(* IEC 61131-3 sources: repolevel_ST_code_completion/dataset/project_code/ProductionLine/FUN, 6 files *)

(* ---- Motor.st ---- *)
FUNCTION_BLOCK Motor
VAR_INPUT
	MotorI:MotorI;
END_VAR
VAR_OUTPUT
	MotorO:MotorO;
END_VAR
VAR
	WaitTimer:TON;
	InternalSequenceDelay:time;
END_VAR

SetFault();
ResetFault();

(* ---- Motor_ResetFault.st ---- *)
METHOD ResetFault : BOOL
VAR_INPUT
	MotorI:MotorI;
END_VAR
VAR_OUTPUT
	MotorO:MotorO;
END_VAR
VAR
	WaitTimer:TON;
	InternalSequenceDelay:time;
	ResetDetect:r_trig;
END_VAR

ResetDetect(CLK:=MotorI.FaultReset);

IF ResetDetect.Q THEN
	MotorO.FaultStatus:=FALSE;
END_IF

(* ---- Motor_SetFault.st ---- *)
METHOD SetFault : BOOL
VAR_INPUT
	MotorI:MotorI;
END_VAR
VAR_OUTPUT
	MotorO:MotorO;
END_VAR
VAR
	WaitTimer:TON;
	InternalSequenceDelay:time;
END_VAR

IF MotorI.Overload THEN
	MotorO.FaultStatus:=TRUE;
	TurnOff();
END_IF

(* ---- Motor_SetWaitTime.st ---- *)
METHOD SetWaitTime : BOOL
VAR_INPUT
	MotorI:MotorI;
	SequenceDelay:TIME;
END_VAR
VAR_OUTPUT
	MotorO:MotorO;
END_VAR
VAR
	WaitTimer:TON;
	InternalSequenceDelay:time;
END_VAR

InternalSequenceDelay:=SequenceDelay;

(* ---- Motor_TurnOff.st ---- *)
METHOD TurnOff : BOOL
VAR_INPUT
	MotorI:MotorI;
END_VAR
VAR_OUTPUT
	MotorO:MotorO;
END_VAR
VAR
	WaitTimer:TON;
	InternalSequenceDelay:time;
END_VAR

MotorO.Coil:=false;

(* ---- Motor_TurnOn.st ---- *)
METHOD TurnOn : BOOL
VAR_INPUT
	MotorI:MotorI;
END_VAR
VAR_OUTPUT
	MotorO:MotorO;
END_VAR
VAR
	WaitTimer:TON;
	InternalSequenceDelay:time;
END_VAR

IF MotorO.FaultStatus = FALSE THEN
	WaitTimer(IN:=TRUE , PT:=InternalSequenceDelay);
END_IF

IF WaitTimer.Q THEN
	MotorO.Coil:=TRUE;
	WaitTimer(IN:=FALSE);
END_IF
